// TIA Portal V15.1 export
// export: Created 2024-05-17T05:38:29.6170665Z, ExportSetting WithDefaults, DisplayName Totally Integrated Automation Portal, DisplayVersion V15.1 Update 5, DisplayName TIA Portal Openness, DisplayVersion V15.1 Update 5, DisplayName SINAMICS Startdrive Advanced, DisplayVersion V15.1, DisplayName G130, G150, S120, S150, SINAMICS MV, S210, DisplayVersion V15.1, DisplayName G110M, G120, G120C, G120D, G120P, DisplayVersion V15.1, DisplayName STEP 7 Professional, DisplayVersion V15.1 Update 5, DisplayName STEP 7 Safety, DisplayVersion V15.1, DisplayName WinCC Professional, DisplayVersion V15.1 Update 5, DisplayName SIMATIC Visualization Architect, DisplayVersion V15.1
FUNCTION_BLOCK "LPNIODiagIPS7-1500"   // FB2211, SCL
{ S7_Optimized_Access := 'TRUE' }
VERSION : 0.1
// stored: AutoNumber false, IsIECCheckEnabled false, IsRetainMemResEnabled false, MemoryReserve 100, SetENOAutomatically False, UDAEnableTagReadback false
   VAR_INPUT
      I_StartFillList { ExternalAccessible := 'False'; ExternalVisible := 'False'; ExternalWritable := 'False'} : Bool;
      I_LastDeviceNumber { ExternalAccessible := 'False'; ExternalVisible := 'False'; ExternalWritable := 'False'} : Int;   // Last Device of ProfiNet System
   END_VAR
   VAR_OUTPUT
      O_Done { ExternalAccessible := 'False'; ExternalVisible := 'False'; ExternalWritable := 'False'} : Bool;
      O_IPAddress { ExternalAccessible := 'False'; ExternalVisible := 'False'; ExternalWritable := 'False'} : Array[0..255] of String[15];
   END_VAR
   VAR_IN_OUT
      IO_DeviceExist : Array[0..255] of Bool;   // IO devices exist
      IO_HWIdentifier : Array[0..255] of UInt;   // HW Device
      IO_GetStationIP : Array[0..255] of IF_CONF_v4;   // Read out Station Information
   END_VAR
   VAR
      Index { ExternalAccessible := 'False'; ExternalVisible := 'False'; ExternalWritable := 'False'} : Int;
      LastDeviceNumber { ExternalAccessible := 'False'; ExternalVisible := 'False'; ExternalWritable := 'False'} : Int;   // Last Device of ProfiNet System
      Done { ExternalAccessible := 'False'; ExternalVisible := 'False'; ExternalWritable := 'False'} : Bool;
      DoneDelay { ExternalAccessible := 'False'; ExternalVisible := 'False'; ExternalWritable := 'False'} : Bool;
      ReturnGetStationInfoBusy_IP { ExternalAccessible := 'False'; ExternalVisible := 'False'; ExternalWritable := 'False'} : Bool;   // Temp
      ReturnGetStationInfoDone_IP { ExternalAccessible := 'False'; ExternalVisible := 'False'; ExternalWritable := 'False'} : Bool;   // Temp
      ReturnGetStationInfoError_IP { ExternalAccessible := 'False'; ExternalVisible := 'False'; ExternalWritable := 'False'} : Bool;   // Temp
      ReturnGetStationInfoStatus_IP { ExternalAccessible := 'False'; ExternalVisible := 'False'; ExternalWritable := 'False'} : Word;   // Temp
      IPAddress_ADDR1 { ExternalAccessible := 'False'; ExternalVisible := 'False'; ExternalWritable := 'False'} : String;
      IPAddress_ADDR2 { ExternalAccessible := 'False'; ExternalVisible := 'False'; ExternalWritable := 'False'} : String;
      IPAddress_ADDR3 { ExternalAccessible := 'False'; ExternalVisible := 'False'; ExternalWritable := 'False'} : String;
      IPAddress_ADDR4 { ExternalAccessible := 'False'; ExternalVisible := 'False'; ExternalWritable := 'False'} : String;
      IPAddress { ExternalAccessible := 'False'; ExternalVisible := 'False'; ExternalWritable := 'False'} : String[15];
      GetStationInfo_IP { ExternalAccessible := 'False'; ExternalVisible := 'False'; ExternalWritable := 'False'; S7_SetPoint := 'True'} : GetStationInfo;   // Get Station
      TimerDone { ExternalAccessible := 'False'; ExternalVisible := 'False'; ExternalWritable := 'False'; S7_SetPoint := 'True'} : TON_TIME;
      EdgeStartFillList { ExternalAccessible := 'False'; ExternalVisible := 'False'; ExternalWritable := 'False'; S7_SetPoint := 'True'} : R_TRIG;
   END_VAR
BEGIN
   #EdgeStartFillList(CLK:=#I_StartFillList);

   IF #EdgeStartFillList.Q THEN
       #Done := False;
       #Index := 0;
   END_IF;

   #LastDeviceNumber := #I_LastDeviceNumber;
   IF #I_LastDeviceNumber < 1 THEN
       #LastDeviceNumber := 1;
   END_IF;
   IF #I_LastDeviceNumber > 254 THEN
       #LastDeviceNumber := 254;
   END_IF;

   #TimerDone(IN := #Done,
              PT := T#500ms,
              Q => #DoneDelay);

   IF (#I_StartFillList & NOT #Done) THEN
       #Index := #Index + 1;
       WHILE (#IO_DeviceExist[#Index] & NOT #ReturnGetStationInfoDone_IP) DO
               #GetStationInfo_IP(REQ := #IO_DeviceExist[#Index] & NOT #ReturnGetStationInfoBusy_IP,
                      LADDR := #IO_HWIdentifier[#Index],
                      MODE := 1,
                      DONE => #ReturnGetStationInfoDone_IP,
                      BUSY => #ReturnGetStationInfoBusy_IP,
                      ERROR => #ReturnGetStationInfoError_IP,
                      STATUS => #ReturnGetStationInfoStatus_IP,
                      DATA := #IO_GetStationIP[#Index]);
        END_WHILE;
        #ReturnGetStationInfoDone_IP := False;

       VAL_STRG(IN := BYTE_TO_USINT(#IO_GetStationIP[#Index].InterfaceAddress.ADDR[1]),
                SIZE := 3,
                PREC := 0,
                FORMAT := 16#0000,
                P := 1,
                OUT => #IPAddress_ADDR1);
       VAL_STRG(IN := BYTE_TO_USINT(#IO_GetStationIP[#Index].InterfaceAddress.ADDR[2]),
                SIZE := 3,
                PREC := 0,
                FORMAT := 16#0000,
                P := 1,
                OUT => #IPAddress_ADDR2);
       VAL_STRG(IN := BYTE_TO_USINT(#IO_GetStationIP[#Index].InterfaceAddress.ADDR[3]),
                SIZE := 3,
                PREC := 0,
                FORMAT := 16#0000,
                P := 1,
                OUT => #IPAddress_ADDR3);
       VAL_STRG(IN := BYTE_TO_USINT(#IO_GetStationIP[#Index].InterfaceAddress.ADDR[4]),
                SIZE := 3,
                PREC := 0,
                FORMAT := 16#0000,
                P := 1,
                OUT => #IPAddress_ADDR4);

       #IPAddress := CONCAT_STRING(IN1 := #IPAddress_ADDR1, IN2 :='.');
       #IPAddress := CONCAT_STRING(IN1 := #IPAddress, IN2 := #IPAddress_ADDR2);
       #IPAddress := CONCAT_STRING(IN1 := #IPAddress, IN2 := '.');
       #IPAddress := CONCAT_STRING(IN1 := #IPAddress, IN2 := #IPAddress_ADDR3);
       #IPAddress := CONCAT_STRING(IN1 := #IPAddress, IN2 := '.');
       #IPAddress := CONCAT_STRING(IN1 := #IPAddress, IN2 := #IPAddress_ADDR4);
       #O_IPAddress[#Index] := #IPAddress;
       IF #Index = #LastDeviceNumber THEN
           #Done := True;
       END_IF;
   END_IF;

   #O_Done := #DoneDelay;
END_FUNCTION_BLOCK
